# EPICS IOC start-up script: test/startup/st.mcu015-pils.iocsh
epicsEnvSet("MOTOR_PORT",      "$(SM_MOTOR_PORT=MCU1)")

epicsEnvSet("IPADDR",          "$(SM_IPADDR=172.30.41.143)")
epicsEnvSet("IPPORT",          "$(SM_IPPORT=48898)")
epicsEnvSet("ASYN_PORT",       "$(SM_ASYN_PORT=MC_CPU1)")
epicsEnvSet("P",               "$(SM_P=LabS-MCAG:MC-MCU-15:)")
epicsEnvSet("R",               "")
epicsEnvSet("PREC",            "$(SM_PREC=3)")
epicsEnvSet("SM_NOAXES",       "2")
epicsEnvSet("ECM_OPTIONS",     "adsPort=852;amsNetIdRemote=172.30.41.143.1.1;amsNetIdLocal=172.30.38.12.1.1"

< ethercatmcController.iocsh

#
# Axis 1
#
epicsEnvSet("AXISCONFIG",      "")
epicsEnvSet("R",               "$(SM_R=m1)")
epicsEnvSet("AXIS_NO",         "$(SM_AXIS_NO=1)")
epicsEnvSet("DESC",            "$(SM_DESC=DESC)")
epicsEnvSet("EGU",             "$(SM_EGU=EGU)")
epicsEnvSet("RAWENCSTEP_ADEL", 0)
epicsEnvSet("RAWENCSTEP_MDEL", 0)
< ethercatmcIndexerAxis.iocsh
< ethercatmcAxisdebug.iocsh

#
# Axis 2
#
epicsEnvSet("AXISCONFIG",      "")
epicsEnvSet("R",               "$(SM_R=m2)")
epicsEnvSet("AXIS_NO",         "$(SM_AXIS_NO=2)")
epicsEnvSet("RAWENCSTEP_ADEL", 0)
epicsEnvSet("RAWENCSTEP_MDEL", 0)
< ethercatmcIndexerAxis.iocsh
< ethercatmcAxisdebug.iocsh
